PROGRAM MAIN
VAR
	bInput : BOOL;
	bOutput : BOOL;
END_VAR

bOutput := bInput;

END_PROGRAM

(* stored: Version 1.1.0.1, ProductVersion 3.1.4024.12
   POU MAIN: Id {628c5be1-be64-4f4a-b2c2-f4ac993c6eab}, SpecialFunc None *)
